Omron CX-Programmer project NewProject (CX-Programmer 9.75)

# PLC Sistem_Kontrol_Air_Limbah: CP1E N20

## Global symbols (name address type ; comment)
0.00 BOOL  ; PB Start
0.01 BOOL  ; PB Stop
0.02 BOOL  ; Maks LVL Sensor
0.03 BOOL  ; Min LVL Sensor
0.04 BOOL  ; Full Pembuangan
0.05 BOOL  ; Low Pembuangan
100.00 BOOL  ; Valve Limbah
100.01 BOOL  ; Valve Air
100.02 BOOL  ; Valve Kuras
100.03 BOOL  ; Mixer
100.04 BOOL  ; Pompa Klorin
100.05 BOOL  ; Blower 1
100.06 BOOL  ; Blower 2
100.07 BOOL  ; Pompa Pembuangan
10.00 BOOL  ; Proses
200.00 BOOL  ; DIFU
20.00 BOOL  ; DIFU Valve Kuras
T000 BOOL  ; Timer 1
T001 BOOL  ; Timer Blower 1
T002 BOOL  ; Timer Blower 2

## Program NewProgram1 (cyclic task 0)

### Section Section1

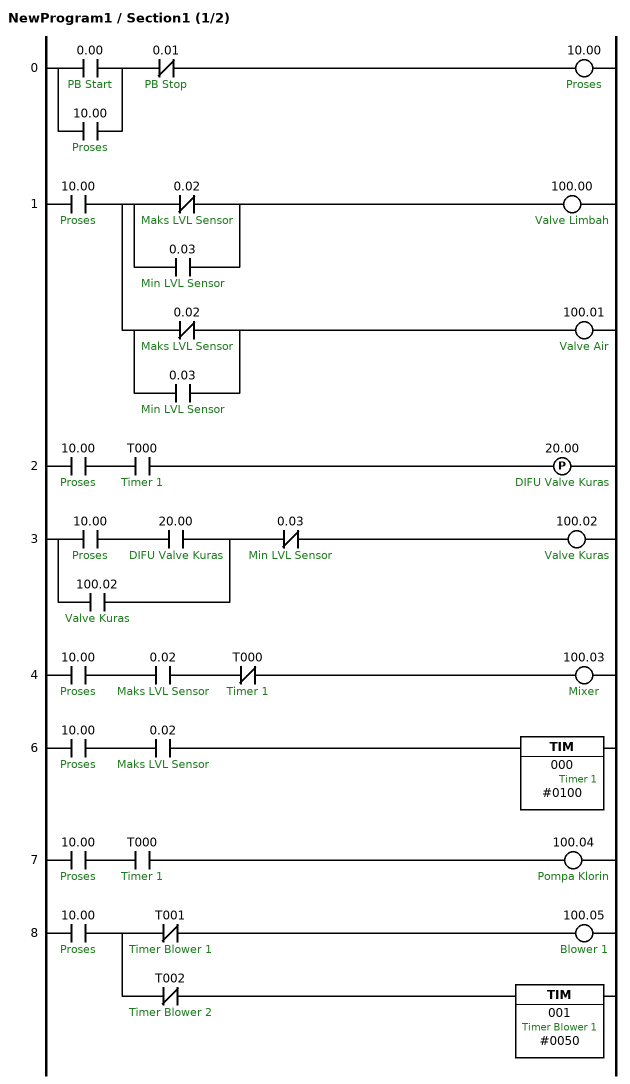
; rung 0
LD 0.00  ; PB Start
OR 10.00  ; Proses
ANDNOT 0.01  ; PB Stop
OUT 10.00  ; Proses
; rung 1
LD 10.00  ; Proses
OUT TR0
LDNOT 0.02  ; Maks LVL Sensor
OR 0.03  ; Min LVL Sensor
ANDLD
OUT 100.00  ; Valve Limbah
LD TR0
LDNOT 0.02  ; Maks LVL Sensor
OR 0.03  ; Min LVL Sensor
ANDLD
OUT 100.01  ; Valve Air
; rung 2
LD 10.00  ; Proses
AND T000  ; Timer 1
DIFU(013) 20.00  ; DIFU Valve Kuras
; rung 3
LD 10.00  ; Proses
AND 20.00  ; DIFU Valve Kuras
OR 100.02  ; Valve Kuras
ANDNOT 0.03  ; Min LVL Sensor
OUT 100.02  ; Valve Kuras
; rung 4
LD 10.00  ; Proses
AND 0.02  ; Maks LVL Sensor
ANDNOT T000  ; Timer 1
OUT 100.03  ; Mixer
; rung 6
LD 10.00  ; Proses
AND 0.02  ; Maks LVL Sensor
TIM 000 #0100  ; Timer 1
; rung 7
LD 10.00  ; Proses
AND T000  ; Timer 1
OUT 100.04  ; Pompa Klorin
; rung 8
LD 10.00  ; Proses
OUT TR0
ANDNOT T001  ; Timer Blower 1
OUT 100.05  ; Blower 1
LD TR0
ANDNOT T002  ; Timer Blower 2
TIM 001 #0050  ; Timer Blower 1

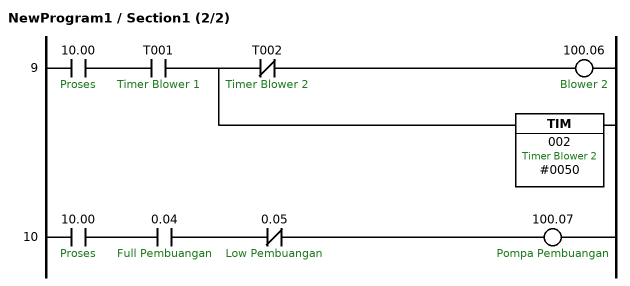
; rung 9
LD 10.00  ; Proses
AND T001  ; Timer Blower 1
OUT TR0
ANDNOT T002  ; Timer Blower 2
OUT 100.06  ; Blower 2
LD TR0
TIM 002 #0050  ; Timer Blower 2
; rung 10
LD 10.00  ; Proses
AND 0.04  ; Full Pembuangan
ANDNOT 0.05  ; Low Pembuangan
OUT 100.07  ; Pompa Pembuangan

### Section END
; rung 0
END(001)